Yaskawa INFORM job: CLEAN-R1.JBI

/JOB
//NAME CLEAN-R1
///FOLDERNAME CLEAN
//POS
///NPOS 9,0,0,0,0,0
///TOOL 0
///POSTYPE PULSE
///PULSE
C00000=1,-80000,-25000,20,-113944,0
C00001=103531,-80000,-25000,20,-113944,0
C00002=98389,-82063,-93533,-21762,-79074,49222
C00003=98704,-79928,-99251,-22171,-74694,49919
C00004=98962,-75779,-101309,-22564,-71477,50449
C00005=98704,-79928,-99251,-22171,-74694,49919
C00006=98389,-82063,-93533,-21762,-79074,49222
C00007=103531,-80000,-25000,20,-113944,0
C00008=1,-80000,-25000,20,-113944,0
//INST
///DATE 2021/10/29 11:50
///ATTR SC,RO
///GROUP1 RB1
NOP
MOVJ C00000 VJ=50.00
MOVJ C00001 VJ=50.00
WAIT IN#(12)=ON
WAIT IN#(15)=ON
MOVJ C00002 VJ=75.00
MOVL C00003 V=211.7
DOUT OT#(4092) ON
MOVL C00004 V=41.7 PL=0
CALL JOB:REAMCYCL
MOVL C00005 V=41.7
DOUT OT#(4092) OFF
MOVJ C00006 VJ=50.00
MOVJ C00007 VJ=75.00
MOVJ C00008 VJ=75.00
SET I001 I000
END
